Fanuc KAREL source: kt00903.KL

PROGRAM KT00903
%STACKSIZE=65535
%PRIORITY=65535
%NOLOCKGROUP
VAR
P1 : POSITION
P2 : POSITION
-- UNRESOLVED DECLARATIONS (source type spelling not recovered)
-- OUT : TYPE_0x0013 (type_u16=0x0013)
BEGIN
OUT=APPROACH(P1)
END KT00903
